// TIA Portal V20 export
TYPE "typeWritePLCData"
   STRUCT
      processData : Bool;
      spareOut_1 : Bool;
      spareOut_2 : Bool;
      spareOut_3 : Bool;
      spareOut_4 : Bool;
      spareOut_5 : Bool;
      spareOut_6 : Bool;
      spareOut_7 : Bool;
      "type" : Int;
      module : Int;
      machine : DInt := 1;
      fixture : Int := 0;
      pun : Array[0..31] of Char;
      unWinderInfeed : "typeStationDataUnwidnerInfeed";
      reelCutInspection : "typeStationDataReelCutInspection";
   END_STRUCT;
END_TYPE
